(* PLC project Tankfil, Unknown Tankfil 1 *)
(* stored: creationDateTime 2026-09-27T11:26:58, modificationDateTime 2026-09-27T13:29:29 *)

PROGRAM TankFill
  VAR
    TankFillAuto_Cmd : BOOL;  (* Internal automatic fill latch/command *)
    TankValveOpen : BOOL;  (* Discrete command/status for the fill valve *)
    Estop_Cmd : BOOL;  (* Emergency-stop input; TRUE forces automatic fill to stop *)
    TankLevelHi_Alarm : BOOL;  (* High-level alarm state *)
    TankLevelLo_Alarm : BOOL;  (* Low-level alarm state *)
    TankLevel_LIT : REAL;  (* Measured tank level in feet *)
    TankEmpty_SP : REAL := 2.0 ft;  (* Automatic fill start setpoint (2.0 ft) *)
    TankFull_SP : REAL := 8.0 ft;  (* Automatic fill stop setpoint (8.0 ft) *)
    TankLoAlarm_SP : REAL := 1.0 ft;  (* Low-level alarm setpoint (1.0 ft) *)
    TankHiAlarm_SP : REAL := 9.0 ft;  (* High-level alarm setpoint (9.0 ft) *)
    TankEmpty : BOOL;  (* Tank is Empty *)
    TankFull : BOOL;  (* Tank is Full *)
    TankHighAlarm : BOOL;
    TankLowAlarm : BOOL;
  END_VAR

(* LD diagram, written out as Structured Text *)
IF TankEmpty THEN TankFillAuto_Cmd := TRUE; END_IF;
IF TankFull THEN TankFillAuto_Cmd := FALSE; END_IF;
IF Estop_Cmd THEN TankFillAuto_Cmd := FALSE; END_IF;
IF TankLevelHi_Alarm THEN TankFillAuto_Cmd := FALSE; END_IF;
TankLevelHi_Alarm := TankHighAlarm;
TankLevelLo_Alarm := TankLowAlarm;
(* drawn but not wired to any output: TankFillAuto_Cmd, TankLevelHi_Alarm *)
END_PROGRAM

CONFIGURATION Config0
  VAR_GLOBAL
    TankFillAuto_Cmd : BOOL;  (* Internal automatic fill latch/command *)
    TankValveOpen : BOOL;  (* Discrete command/status for the fill valve *)
    Estop_Cmd : BOOL;  (* Emergency-stop input; TRUE forces automatic fill to stop *)
    TankLevelHi_Alarm : BOOL;  (* High-level alarm state *)
    TankLevelLo_Alarm : BOOL;  (* Low-level alarm state *)
    TankLevel_LIT : REAL;  (* Measured tank level in feet *)
    TankEmpty_SP : REAL := 2.0 ft;  (* Automatic fill start setpoint (2.0 ft) *)
    TankFull_SP : REAL := 8.0 ft;  (* Automatic fill stop setpoint (8.0 ft) *)
    TankLoAlarm_SP : REAL := 1.0 ft;  (* Low-level alarm setpoint (1.0 ft) *)
    TankHiAlarm_SP : REAL := 9.0 ft;  (* High-level alarm setpoint (9.0 ft) *)
  END_VAR
  RESOURCE Res0 ON PLC
    TASK task0(INTERVAL := T#20ms, PRIORITY := 0);
    PROGRAM instance0 WITH task0 : TankFill;
  END_RESOURCE
END_CONFIGURATION
